FUNCTION_BLOCK FB_BaseUnit IMPLEMENTS I_ResourceLock
VAR
	// Owner ID zero means that no Service currently owns this BaseUnit.
	_ResourceOwnerId : T_ResourceOwnerId;
END_VAR

METHOD PUBLIC FINAL M_AcquireResource : BOOL
VAR_INPUT
	OwnerId : T_ResourceOwnerId;
END_VAR
// Reject zero because it represents the unowned state.
M_AcquireResource := FALSE;
IF OwnerId = 0 THEN
	RETURN;
END_IF

// Re-acquiring with the current Owner ID is intentionally idempotent.
IF (_ResourceOwnerId = 0) OR (_ResourceOwnerId = OwnerId) THEN
	_ResourceOwnerId := OwnerId;
	M_AcquireResource := TRUE;
END_IF
END_METHOD

METHOD PUBLIC FINAL M_IsResourceOwner : BOOL
VAR_INPUT
	OwnerId : T_ResourceOwnerId;
END_VAR
// Zero can never identify a valid Resource Owner.
M_IsResourceOwner := (OwnerId <> 0) AND (_ResourceOwnerId = OwnerId);
END_METHOD

METHOD PUBLIC FINAL M_ReleaseResource : BOOL
VAR_INPUT
	OwnerId : T_ResourceOwnerId;
END_VAR
// Only the current Owner may release the Resource.
M_ReleaseResource := FALSE;
IF NOT M_IsResourceOwner(OwnerId := OwnerId) THEN
	RETURN;
END_IF

_ResourceOwnerId := 0;
M_ReleaseResource := TRUE;
END_METHOD

PROPERTY PUBLIC FINAL ResourceIsAcquired : BOOL
GET
ResourceIsAcquired := _ResourceOwnerId <> 0;
END_GET
END_PROPERTY

PROPERTY PUBLIC FINAL ResourceOwnerId : T_ResourceOwnerId
GET
ResourceOwnerId := _ResourceOwnerId;
END_GET
END_PROPERTY

END_FUNCTION_BLOCK

(* stored: Version 1.1.0.1, ProductVersion 3.1.4026.18
   POU FB_BaseUnit: Id {f4702b47-ca2c-49e4-bf41-fa6124c0142b}, SpecialFunc None
   Method M_AcquireResource: Id {cdbf4753-4286-4f58-8516-80dd542d86d2}
   Method M_IsResourceOwner: Id {8401a888-1361-4392-8830-38d11946572d}
   Method M_ReleaseResource: Id {16d09c57-8934-4d9d-88e3-8d43c058994d}
   Property ResourceIsAcquired: Id {f5b55c57-27a4-4fc0-896e-8ed3ee28765f}
   Get Get: Id {e5ed7dea-a104-41a6-8134-c1442b588d98}
   Property ResourceOwnerId: Id {7fb00a7d-6329-4361-873e-1ef67de1777d}
   Get Get: Id {3f67c5dc-572d-499f-bb86-cf0ab802adbc} *)
